TYPE Udt_ParLog_Old :
STRUCT
	ParList		: ARRAY [0..GVL_Parameters.MAX_PARAMETERS] OF Udt_Parameter_2 ; // active parameter list
END_STRUCT
END_TYPE

(* stored: Version 1.1.0.1, ProductVersion 3.1.4024.4
   DUT Udt_ParLog_Old: Id {2c3e3688-0d27-4d22-b1da-a5bd1c07683d} *)
